TYPE ST_HmiBottomBar :
STRUCT CONSTANT
	Start					: STRING := 'WebContent/Bottom/NavigationBarStart.content';
	Alarm					: STRING := 'WebContent/Bottom/NavigationBarAlarm.content';
	General_ReturnToStart	: STRING := 'WebContent/Bottom/NavigationBarReturnToStart.content';
END_STRUCT
END_TYPE

(* stored: Version 1.1.0.1, ProductVersion 3.1.4024.12
   DUT ST_HmiBottomBar: Id {31e56192-536d-49be-b77c-f613bc4b327d} *)
